FUNCTION_BLOCK EL3112
VAR
	_io : EL3xx2_Data;
	{attribute addProperty Name "WcState"}
	_wcState : WcStateInputToggle;
	{attribute addProperty Name "Info data"}
	_infoData : InfoDataAds;
END_VAR

PROPERTY IO : REFERENCE TO EL3xx2_Data
GET
IO REF= _io;
END_GET
END_PROPERTY

PROPERTY WcState : REFERENCE TO WcStateInputToggle
GET
WcState REF= _wcState;
END_GET
END_PROPERTY

END_FUNCTION_BLOCK

(* stored: Version 1.1.0.1, ProductVersion 3.1.4024.9
   POU EL3112: Id {27dc09c2-e8d3-0be5-1fb8-7ef7e30876ea}, SpecialFunc None
   Property IO: Id {a215d5ab-32e4-09bc-3516-b6eb828c0880}
   Get Get: Id {f83b8b89-9662-0e92-0ee7-7496d016d0be}
   Property WcState: Id {d3febc3f-0c19-0c56-19c3-905df4f93a7e}
   Get Get: Id {9aec69bd-53a5-0340-2c21-1c1f5aa99fe0} *)
